{attribute 'GeneratedUsingTerminal: EL6201-0000-0017'}
{attribute addProperty BoxType "EL6201-0000-0017"}
{attribute addProperty Id "Slave_23A_DO0BOOL1Slave_23A_DO1BOOL1Slave_23A_DO2BOOL1Slave_23A_DO3BOOL1Slave_23B_DO0BOOL1Slave_23B_DO1BOOL1Slave_23B_DO2BOOL1Slave_23B_DO3BOOL1"}
{attribute addProperty CRC "3921656996"}
{attribute addProperty Size "8"}
TYPE Slave_23_Outputs_E9BFBCA4 :
STRUCT
	{attribute addProperty Name "Slave_23A_DO0"}
	Slave_23A_DO0 : BOOL;
	{attribute addProperty Name "Slave_23A_DO1"}
	Slave_23A_DO1 : BOOL;
	{attribute addProperty Name "Slave_23A_DO2"}
	Slave_23A_DO2 : BOOL;
	{attribute addProperty Name "Slave_23A_DO3"}
	Slave_23A_DO3 : BOOL;
	{attribute addProperty Name "Slave_23B_DO0"}
	Slave_23B_DO0 : BOOL;
	{attribute addProperty Name "Slave_23B_DO1"}
	Slave_23B_DO1 : BOOL;
	{attribute addProperty Name "Slave_23B_DO2"}
	Slave_23B_DO2 : BOOL;
	{attribute addProperty Name "Slave_23B_DO3"}
	Slave_23B_DO3 : BOOL;
END_STRUCT
END_TYPE

(* stored: Version 1.2.0.0, ProductVersion 3.1.4024.9
   DUT Slave_23_Outputs_E9BFBCA4: Id {14e48e6d-62a4-495a-8132-097c1f99456e} *)
